PROGRAM prgCom
VAR
	fbCom			: FB_MqttCommunicator_V3;
END_VAR

fbCom(
	bConnect:= TRUE,
	strAuthKey:= 'TSG88376368072',
	sUserName:= 'ab6b7704-0b2c-4c94-8e47-13d25c5f2bfa', 
	sUserPassword:= '78b266a9-af78-4bf8-8bad-800f54d6b5e5', 
	eSavePositionCertificate:= eSavePositionOnPLC.ePostionC, 
	bConnected=> , 
	bError=> , 
	hrErrorCode=> , 
	eConnectionState=> , 
	eErrorMessage_Out=> );

END_PROGRAM

(* stored: Version 1.1.0.1, ProductVersion 3.1.4024.12
   POU prgCom: Id {ab2e2113-e5ef-4576-b3e1-d9e4709b48fc}, SpecialFunc None *)
